Yaskawa INFORM job: frame_cylinder_program.JBI

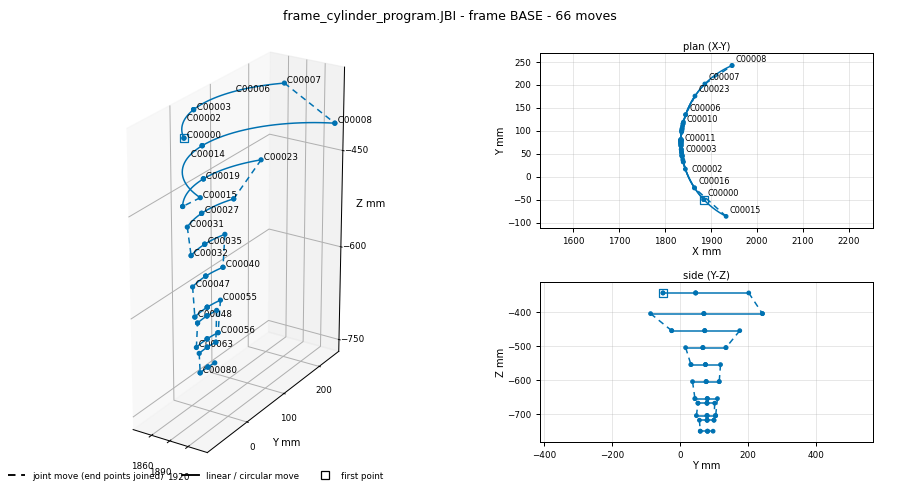
[picture p0: tool path of frame_cylinder_program.JBI in frame BASE, 66 of 91 moves have a stored position in this frame; points joined in program order, loops and branches not executed]
/JOB
//NAME frame_cylinder_program
//POS
///NPOS 88,0,88,0,0,0
///TOOL 0
///POSTYPE BASE
///RECTAN
///RCONF 0,0,0,0,0,0,0,0,0,0,0,0,0,0,0,0,0,0,0,0,0,0,0,0
C00000=1884.394542,-50.031083,-343.694000,-136.509314,-89.999999,5.000000
C00001=1884.394542,-50.031083,-343.694000,-136.509314,-89.999999,5.000000
C00002=1850.144326,1.312380,-343.694000,-156.077737,-90.000000,5.000000
C00003=1836.859115,46.048801,-343.694000,-170.842969,-89.999999,5.000000
C00004=1836.859115,46.048801,-343.694000,-170.842969,-89.999999,5.000000
C00005=1836.859115,46.048801,-343.694000,-170.842969,-89.999999,5.000000
C00006=1844.518969,134.302120,-343.694000,160.921978,-90.000000,5.000000
C00007=1886.628193,202.239457,-343.694000,135.494726,-90.000000,5.000000
C00008=1946.006368,242.451329,-404.545000,112.718275,-90.000000,5.000000
C00009=1946.006368,242.451329,-404.545000,112.718275,-90.000000,5.000000
C00010=1838.207828,111.236876,-404.545000,168.472458,-90.000000,5.000000
C00011=1834.605264,70.264949,-404.545000,-175.000000,-89.999999,5.000000
C00012=1834.605264,70.264949,-404.545000,-175.000000,-89.999999,5.000000
C00013=1834.605264,70.264949,-404.545000,-175.000000,-89.999999,5.000000
C00014=1841.409166,25.491669,-404.545000,-164.196114,-89.999999,5.000000
C00015=1933.037215,-86.515147,-404.545000,-117.233587,-90.000000,5.000000
C00016=1864.129951,-24.398180,-454.675000,-146.833044,-90.000000,5.000000
C00017=1864.129951,-24.398180,-454.675000,-146.833044,-90.000000,5.000000
C00018=1838.665966,36.480281,-454.675000,-167.770204,-90.000000,5.000000
C00019=1834.557333,72.820909,-454.675000,-175.000000,-90.000000,5.000000
C00020=1834.557333,72.820909,-454.675000,-175.000000,-90.000000,5.000000
C00021=1834.557333,72.820909,-454.675000,-175.000000,-90.000000,5.000000
C00022=1837.076075,105.161599,-454.675000,170.422390,-89.999999,5.000000
C00023=1865.127032,175.802530,-454.675000,146.262336,-90.000000,5.000000
C00024=1844.824577,135.178503,-504.569000,160.629133,-90.000000,5.000000
C00025=1844.824577,135.178503,-504.569000,160.629133,-90.000000,5.000000
C00026=1835.671829,95.147144,-504.569000,173.613458,-89.999999,5.000000
C00027=1834.704334,67.339296,-504.569000,-175.000000,-90.000000,5.000000
C00028=1834.704334,67.339296,-504.569000,-175.000000,-90.000000,5.000000
C00029=1834.704334,67.339296,-504.569000,-175.000000,-90.000000,5.000000
C00030=1838.046230,39.459863,-504.569000,-168.730447,-89.999999,5.000000
C00031=1844.189438,16.554590,-504.569000,-161.242676,-90.000000,5.000000
C00032=1839.636807,32.246486,-554.489000,-166.399661,-90.000000,5.000000
C00033=1839.636807,32.246486,-554.489000,-166.399661,-90.000000,5.000000
C00034=1835.839875,53.299356,-554.489000,-173.153301,-90.000000,5.000000
C00035=1834.544890,74.884417,-554.489000,-175.000000,-90.000000,5.000000
C00036=1834.544890,74.884417,-554.489000,-175.000000,-90.000000,5.000000
C00037=1834.544890,74.884417,-554.489000,-175.000000,-90.000000,5.000000
C00038=1835.510818,93.652721,-554.489000,174.087706,-90.000000,5.000000
C00039=1840.025746,119.225471,-554.489000,165.887251,-89.999999,5.000000
C00040=1839.101763,115.373180,-604.584000,167.137217,-90.000000,5.000000
C00041=1839.101763,115.373180,-604.584000,167.137217,-90.000000,5.000000
C00042=1835.414865,92.701728,-604.584000,174.389285,-90.000000,5.000000
C00043=1834.556573,77.008388,-604.584000,175.000000,-89.999999,5.000000
C00044=1834.556573,77.008388,-604.584000,175.000000,-89.999999,5.000000
C00045=1834.556573,77.008388,-604.584000,175.000000,-89.999999,5.000000
C00046=1835.264894,58.792719,-604.584000,-174.896093,-90.000000,5.000000
C00047=1838.579555,36.881132,-604.584000,-167.899585,-89.999999,5.000000
C00048=1837.194888,44.037704,-654.571500,-170.199645,-89.999999,5.000000
C00049=1837.194888,44.037704,-654.571500,-170.199645,-89.999999,5.000000
C00050=1834.847172,64.473963,-654.571500,-175.000000,-90.000000,5.000000
C00051=1834.622635,80.261125,-654.571500,175.000000,-89.999999,5.000000
C00052=1834.622635,80.261125,-654.571500,175.000000,-89.999999,5.000000
C00053=1834.622635,80.261125,-654.571500,175.000000,-89.999999,5.000000
C00054=1835.520179,93.742899,-654.571500,174.059100,-90.000000,5.000000
C00055=1837.979029,110.096412,-654.571500,168.839465,-89.999999,5.000000
C00056=1837.039092,104.941602,-704.574000,170.492777,-90.000000,5.000000
C00057=1837.039092,104.941602,-704.574000,170.492777,-90.000000,5.000000
C00058=1835.365833,92.195332,-704.574000,174.549810,-90.000000,5.000000
C00059=1834.603934,79.578409,-704.574000,175.000000,-90.000000,5.000000
C00060=1834.603934,79.578409,-704.574000,175.000000,-90.000000,5.000000
C00061=1834.603934,79.578409,-704.574000,175.000000,-90.000000,5.000000
C00062=1834.804637,65.238185,-704.574000,-175.000000,-90.000000,5.000000
C00063=1836.510775,48.299533,-704.574000,-171.561576,-90.000000,5.000000
C00064=1835.895600,52.840193,-667.992960,-175.000000,-60.000000,6.992636
C00065=1835.895600,52.840193,-667.992960,-175.000000,-60.000000,6.992636
C00066=1834.737345,66.589147,-667.992960,175.000000,-60.000000,5.000000
C00067=1834.601758,79.492297,-667.992960,-175.000000,-60.000000,-5.000000
C00068=1834.601758,79.492297,-667.992960,-175.000000,-60.000000,-5.000000
C00069=1834.601758,79.492297,-667.992960,-175.000000,-60.000000,-5.000000
C00070=1835.254953,90.990790,-667.992960,-175.000000,-60.000000,-5.068528
C00071=1836.589100,102.118388,-667.992960,175.000000,-60.000000,-8.605194
C00072=1836.275152,99.955912,-718.030460,-175.000000,-60.000000,-7.915736
C00073=1836.275152,99.955912,-718.030460,-175.000000,-60.000000,-7.915736
C00074=1835.110109,89.264153,-718.030460,175.000000,-60.000000,-5.000000
C00075=1834.610524,79.829902,-718.030460,175.000000,-60.000000,-5.000000
C00076=1834.610524,79.829902,-718.030460,175.000000,-60.000000,-5.000000
C00077=1834.610524,79.829902,-718.030460,175.000000,-60.000000,-5.000000
C00078=1834.646095,68.885442,-718.030460,175.000000,-60.000000,5.000000
C00079=1835.419254,57.148853,-718.030460,175.000000,-60.000000,5.624860
C00080=1835.188601,59.670954,-750.392960,-175.000000,-60.000000,5.000000
C00081=1835.188601,59.670954,-750.392960,-175.000000,-60.000000,5.000000
C00082=1834.615234,69.893209,-750.392960,175.000000,-60.000000,5.000000
C00083=1834.643754,80.939270,-750.392960,175.000000,-60.000000,-5.000000
C00084=1834.643754,80.939270,-750.392960,175.000000,-60.000000,-5.000000
C00085=1834.643754,80.939270,-750.392960,175.000000,-60.000000,-5.000000
C00086=1835.157861,89.855660,-750.392960,175.000000,-60.000000,-5.000000
C00087=1835.928417,97.320938,-750.392960,175.000000,-60.000000,-7.077179
///POSTYPE PULSE
///PULSE
EX00000=271360.0
///POSTYPE PULSE
///PULSE
EC00000=271360.0
EC00001=271360.0
EC00002=271360.0
EC00003=271360.0
EC00004=271360.0
EC00005=271360.0
EC00006=271360.0
EC00007=271360.0
EC00008=271360.0
EC00009=271360.0
EC00010=271360.0
EC00011=271360.0
EC00012=271360.0
EC00013=271360.0
EC00014=271360.0
EC00015=271360.0
EC00016=271360.0
EC00017=271360.0
EC00018=271360.0
EC00019=271360.0
EC00020=271360.0
EC00021=271360.0
EC00022=271360.0
EC00023=271360.0
EC00024=271360.0
EC00025=271360.0
EC00026=271360.0
EC00027=271360.0
EC00028=271360.0
EC00029=271360.0
EC00030=271360.0
EC00031=271360.0
EC00032=271360.0
EC00033=271360.0
EC00034=271360.0
EC00035=271360.0
EC00036=271360.0
EC00037=271360.0
EC00038=271360.0
EC00039=271360.0
EC00040=271360.0
EC00041=271360.0
EC00042=271360.0
EC00043=271360.0
EC00044=271360.0
EC00045=271360.0
EC00046=271360.0
EC00047=271360.0
EC00048=271360.0
EC00049=271360.0
EC00050=271360.0
EC00051=271360.0
EC00052=271360.0
EC00053=271360.0
EC00054=271360.0
EC00055=271360.0
EC00056=271360.0
EC00057=271360.0
EC00058=271360.0
EC00059=271360.0
EC00060=271360.0
EC00061=271360.0
EC00062=271360.0
EC00063=271360.0
EC00064=271360.0
EC00065=271360.0
EC00066=271360.0
EC00067=271360.0
EC00068=271360.0
EC00069=271360.0
EC00070=271360.0
EC00071=271360.0
EC00072=271360.0
EC00073=271360.0
EC00074=271360.0
EC00075=271360.0
EC00076=271360.0
EC00077=271360.0
EC00078=271360.0
EC00079=271360.0
EC00080=271360.0
EC00081=271360.0
EC00082=271360.0
EC00083=271360.0
EC00084=271360.0
EC00085=271360.0
EC00086=271360.0
EC00087=271360.0
//INST
///DATE 2023/08/16 15:18
///ATTR SC,RW,RJ
////FRAME BASE
///GROUP1 RB1,ST1
NOP
MOVJ P009 EX000 VJ=15.00
MOVJ C00000 EC00000 VJ=15.0
CALL JOB:SPYON
MOVC C00001 EC00001 V=150.0
MOVC C00002 EC00002 V=150.0
MOVC C00003 EC00003 V=150.0
MOVJ C00004 EC00004 VJ=15.0
MOVC C00005 EC00005 V=150.0
MOVC C00006 EC00006 V=150.0
MOVC C00007 EC00007 V=150.0
MOVJ C00008 EC00008 VJ=15.0
MOVC C00009 EC00009 V=150.0
MOVC C00010 EC00010 V=150.0
MOVC C00011 EC00011 V=150.0
MOVJ C00012 EC00012 VJ=15.0
MOVC C00013 EC00013 V=150.0
MOVC C00014 EC00014 V=150.0
MOVC C00015 EC00015 V=150.0
MOVJ C00016 EC00016 VJ=15.0
MOVC C00017 EC00017 V=150.0
MOVC C00018 EC00018 V=150.0
MOVC C00019 EC00019 V=150.0
MOVJ C00020 EC00020 VJ=15.0
MOVC C00021 EC00021 V=150.0
MOVC C00022 EC00022 V=150.0
MOVC C00023 EC00023 V=150.0
MOVJ C00024 EC00024 VJ=15.0
MOVC C00025 EC00025 V=150.0
MOVC C00026 EC00026 V=150.0
MOVC C00027 EC00027 V=150.0
MOVJ C00028 EC00028 VJ=15.0
MOVC C00029 EC00029 V=150.0
MOVC C00030 EC00030 V=150.0
MOVC C00031 EC00031 V=150.0
MOVJ C00032 EC00032 VJ=15.0
MOVC C00033 EC00033 V=150.0
MOVC C00034 EC00034 V=150.0
MOVC C00035 EC00035 V=150.0
MOVJ C00036 EC00036 VJ=15.0
MOVC C00037 EC00037 V=150.0
MOVC C00038 EC00038 V=150.0
MOVC C00039 EC00039 V=150.0
MOVJ C00040 EC00040 VJ=15.0
MOVC C00041 EC00041 V=150.0
MOVC C00042 EC00042 V=150.0
MOVC C00043 EC00043 V=150.0
MOVJ C00044 EC00044 VJ=15.0
MOVC C00045 EC00045 V=150.0
MOVC C00046 EC00046 V=150.0
MOVC C00047 EC00047 V=150.0
MOVJ C00048 EC00048 VJ=15.0
MOVC C00049 EC00049 V=150.0
MOVC C00050 EC00050 V=150.0
MOVC C00051 EC00051 V=150.0
MOVJ C00052 EC00052 VJ=15.0
MOVC C00053 EC00053 V=150.0
MOVC C00054 EC00054 V=150.0
MOVC C00055 EC00055 V=150.0
MOVJ C00056 EC00056 VJ=15.0
MOVC C00057 EC00057 V=150.0
MOVC C00058 EC00058 V=150.0
MOVC C00059 EC00059 V=150.0
MOVJ C00060 EC00060 VJ=15.0
MOVC C00061 EC00061 V=150.0
MOVC C00062 EC00062 V=150.0
MOVC C00063 EC00063 V=150.0
MOVJ C00064 EC00064 VJ=15.0
MOVC C00065 EC00065 V=150.0
MOVC C00066 EC00066 V=150.0
MOVC C00067 EC00067 V=150.0
MOVJ C00068 EC00068 VJ=15.0
MOVC C00069 EC00069 V=150.0
MOVC C00070 EC00070 V=150.0
MOVC C00071 EC00071 V=150.0
MOVJ C00072 EC00072 VJ=15.0
MOVC C00073 EC00073 V=150.0
MOVC C00074 EC00074 V=150.0
MOVC C00075 EC00075 V=150.0
MOVJ C00076 EC00076 VJ=15.0
MOVC C00077 EC00077 V=150.0
MOVC C00078 EC00078 V=150.0
MOVC C00079 EC00079 V=150.0
MOVJ C00080 EC00080 VJ=15.0
MOVC C00081 EC00081 V=150.0
MOVC C00082 EC00082 V=150.0
MOVC C00083 EC00083 V=150.0
MOVJ C00084 EC00084 VJ=15.0
MOVC C00085 EC00085 V=150.0
MOVC C00086 EC00086 V=150.0
MOVC C00087 EC00087 V=150.0
CALL JOB:SPYOF
MOVJ P009 VJ=15.00
MOVL P009 EX00000 V=150.0
END
